PROGRAM PIST_CYCLE
VAR
	bFirstRun:BOOL:=FALSE;
	counter :INT;
END_VAR


IF NOT bFirstRun THEN
	FOR counter:=1 TO iNUMBER_OF_PISTONS BY 1 DO
		fbPist[counter].bInit:=1;
	END_FOR;
bFirstRun:=TRUE;
END_IF
 

feeder();
clean();
extract();
drop();

ACTION clean:
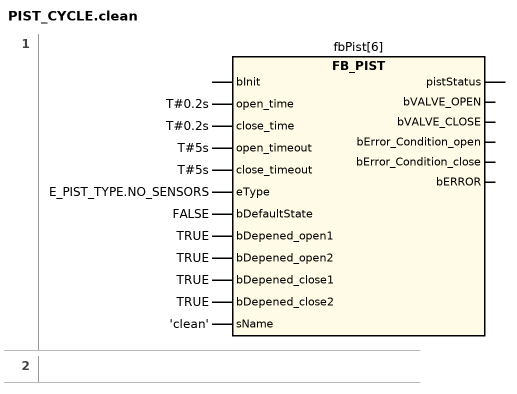
// NETWORK 1
fbPist[6](
    open_time := T#0.2s,
    close_time := T#0.2s,
    open_timeout := T#5s,
    close_timeout := T#5s,
    eType := E_PIST_TYPE.NO_SENSORS,
    bDefaultState := FALSE,
    bDepened_open1 := TRUE,
    bDepened_open2 := TRUE,
    bDepened_close1 := TRUE,
    bDepened_close2 := TRUE,
    sName := 'clean'); // FB_PIST

// NETWORK 2
END_ACTION

ACTION drop:
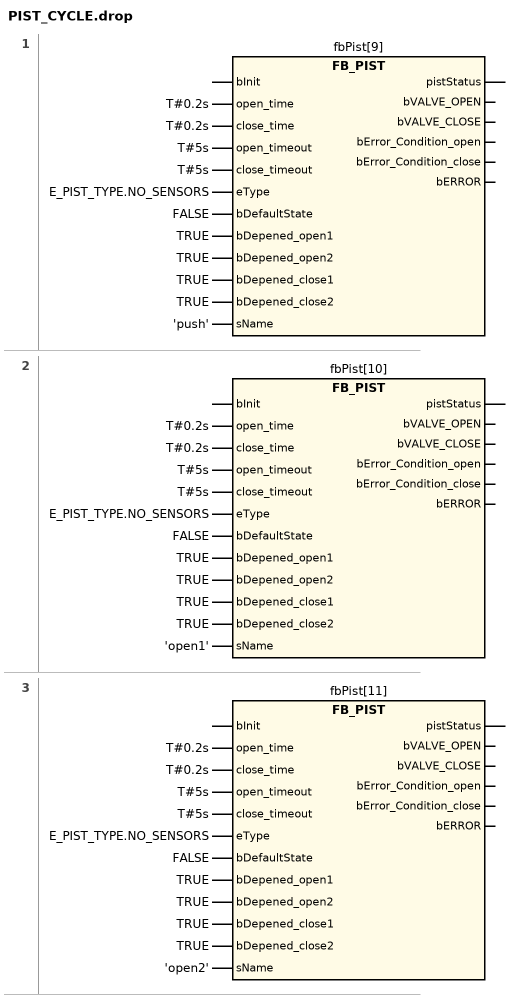
// NETWORK 1
fbPist[9](
    open_time := T#0.2s,
    close_time := T#0.2s,
    open_timeout := T#5s,
    close_timeout := T#5s,
    eType := E_PIST_TYPE.NO_SENSORS,
    bDefaultState := FALSE,
    bDepened_open1 := TRUE,
    bDepened_open2 := TRUE,
    bDepened_close1 := TRUE,
    bDepened_close2 := TRUE,
    sName := 'push'); // FB_PIST

// NETWORK 2
fbPist[10](
    open_time := T#0.2s,
    close_time := T#0.2s,
    open_timeout := T#5s,
    close_timeout := T#5s,
    eType := E_PIST_TYPE.NO_SENSORS,
    bDefaultState := FALSE,
    bDepened_open1 := TRUE,
    bDepened_open2 := TRUE,
    bDepened_close1 := TRUE,
    bDepened_close2 := TRUE,
    sName := 'open1'); // FB_PIST

// NETWORK 3
fbPist[11](
    open_time := T#0.2s,
    close_time := T#0.2s,
    open_timeout := T#5s,
    close_timeout := T#5s,
    eType := E_PIST_TYPE.NO_SENSORS,
    bDefaultState := FALSE,
    bDepened_open1 := TRUE,
    bDepened_open2 := TRUE,
    bDepened_close1 := TRUE,
    bDepened_close2 := TRUE,
    sName := 'open2'); // FB_PIST
END_ACTION

ACTION extract:
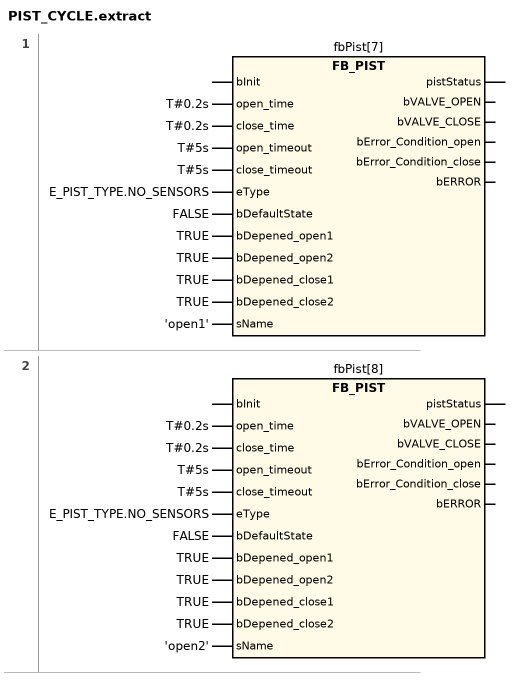
// NETWORK 1
fbPist[7](
    open_time := T#0.2s,
    close_time := T#0.2s,
    open_timeout := T#5s,
    close_timeout := T#5s,
    eType := E_PIST_TYPE.NO_SENSORS,
    bDefaultState := FALSE,
    bDepened_open1 := TRUE,
    bDepened_open2 := TRUE,
    bDepened_close1 := TRUE,
    bDepened_close2 := TRUE,
    sName := 'open1'); // FB_PIST

// NETWORK 2
fbPist[8](
    open_time := T#0.2s,
    close_time := T#0.2s,
    open_timeout := T#5s,
    close_timeout := T#5s,
    eType := E_PIST_TYPE.NO_SENSORS,
    bDefaultState := FALSE,
    bDepened_open1 := TRUE,
    bDepened_open2 := TRUE,
    bDepened_close1 := TRUE,
    bDepened_close2 := TRUE,
    sName := 'open2'); // FB_PIST
END_ACTION

ACTION feeder:
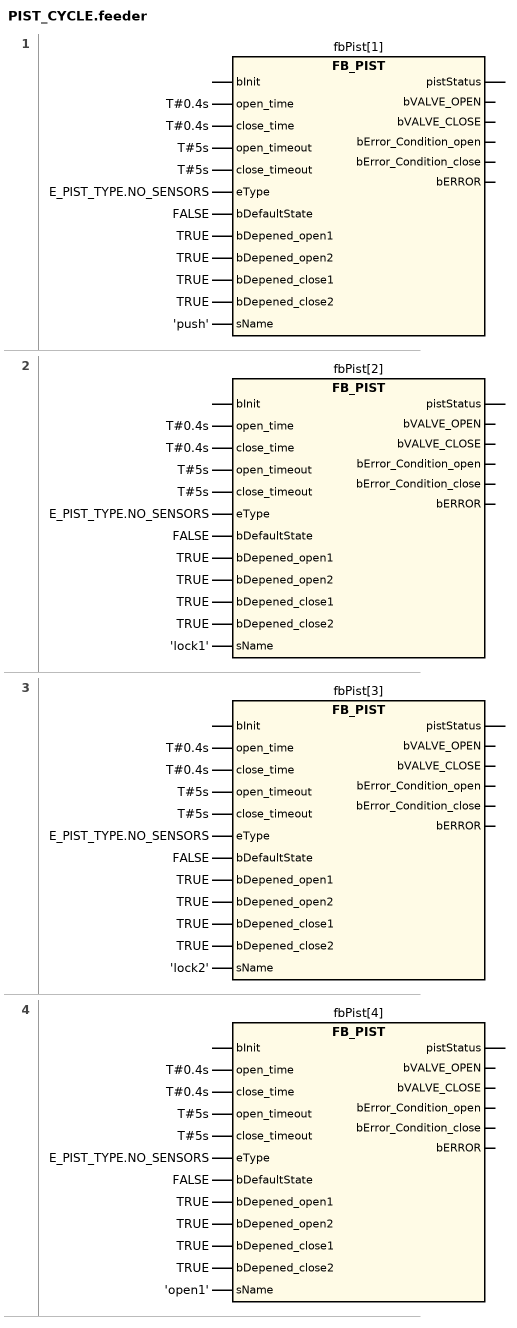
// NETWORK 1
fbPist[1](
    open_time := T#0.4s,
    close_time := T#0.4s,
    open_timeout := T#5s,
    close_timeout := T#5s,
    eType := E_PIST_TYPE.NO_SENSORS,
    bDefaultState := FALSE,
    bDepened_open1 := TRUE,
    bDepened_open2 := TRUE,
    bDepened_close1 := TRUE,
    bDepened_close2 := TRUE,
    sName := 'push'); // FB_PIST

// NETWORK 2
fbPist[2](
    open_time := T#0.4s,
    close_time := T#0.4s,
    open_timeout := T#5s,
    close_timeout := T#5s,
    eType := E_PIST_TYPE.NO_SENSORS,
    bDefaultState := FALSE,
    bDepened_open1 := TRUE,
    bDepened_open2 := TRUE,
    bDepened_close1 := TRUE,
    bDepened_close2 := TRUE,
    sName := 'lock1'); // FB_PIST

// NETWORK 3
fbPist[3](
    open_time := T#0.4s,
    close_time := T#0.4s,
    open_timeout := T#5s,
    close_timeout := T#5s,
    eType := E_PIST_TYPE.NO_SENSORS,
    bDefaultState := FALSE,
    bDepened_open1 := TRUE,
    bDepened_open2 := TRUE,
    bDepened_close1 := TRUE,
    bDepened_close2 := TRUE,
    sName := 'lock2'); // FB_PIST

// NETWORK 4
fbPist[4](
    open_time := T#0.4s,
    close_time := T#0.4s,
    open_timeout := T#5s,
    close_timeout := T#5s,
    eType := E_PIST_TYPE.NO_SENSORS,
    bDefaultState := FALSE,
    bDepened_open1 := TRUE,
    bDepened_open2 := TRUE,
    bDepened_close1 := TRUE,
    bDepened_close2 := TRUE,
    sName := 'open1'); // FB_PIST

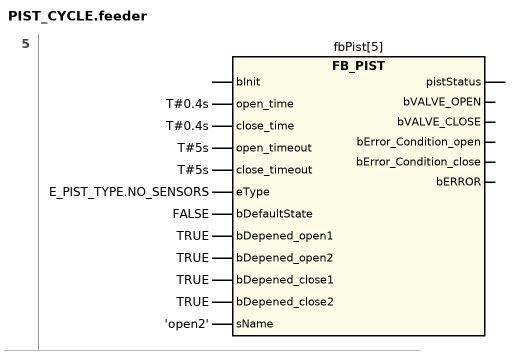
// NETWORK 5
fbPist[5](
    open_time := T#0.4s,
    close_time := T#0.4s,
    open_timeout := T#5s,
    close_timeout := T#5s,
    eType := E_PIST_TYPE.NO_SENSORS,
    bDefaultState := FALSE,
    bDepened_open1 := TRUE,
    bDepened_open2 := TRUE,
    bDepened_close1 := TRUE,
    bDepened_close2 := TRUE,
    sName := 'open2'); // FB_PIST
END_ACTION

END_PROGRAM

(* stored: Version 1.1.0.1, ProductVersion 3.1.4024.12
   POU PIST_CYCLE: Id {b09e4efb-d7ec-45c6-bc50-8222237b347f}, SpecialFunc None
   Action clean: Id {b6db8f46-a5cd-4841-b2f4-af5cb236d344}
   Action drop: Id {b557402b-1722-4c09-8921-9656948ea629}
   Action extract: Id {757442cf-a264-441b-9150-4d5ec0d532ad}
   Action feeder: Id {79acaad4-db77-45ac-865d-5acedade637c} *)
